# EPICS substitutions: tprTriggerApp/Db/pcieSlave_tprTrig.substitutions
# pcieSlave_tprTrig.substitutions

file "tprChannelEvent.db" {
    pattern {        NN    }
            {      "00"    }
            {      "01"    }
            {      "02"    }
            {      "03"    }
            {      "04"    }
            {      "05"    }
            {      "06"    }
            {      "07"    }
            {      "08"    }
            {      "09"    }
            {      "10"    }
            {      "11"    }
}
